// TIA Portal V20 export
DATA_BLOCK "DB_GestionSafetyGate"   // DB202
// stored: AutoNumber false, InstanceOfName FB_GestionSafetyGate, InstanceOfType FB
"FB_GestionSafetyGate"
   // VAR
   //    sExtGate { S7_SetPoint := 'True'} : "FB_CmdCylinder";
   //    sIntGate { S7_SetPoint := 'True'} : "FB_CmdCylinder";
   //    sExtGateCloseCmd : Bool;
   //    sExtGateOpenCmd : Bool;
   //    sIntGateCloseCmd : Bool;
   //    sIntGateOpenCmd : Bool;
   //    sJOG_Cmd : Bool;
   //    sRT_RefCmd : R_TRIG;
   //    sFT_RefCmd : F_TRIG;
   //    sExtGateOpenReq : Bool;
   //    sIntGateOpenReq : Bool;
   //    sExtGateOpened : Bool;
   //    sExtGateClosed : Bool;
   //    sIntGateOpened : Bool;
   //    sIntGateClosed : Bool;
   //    sWaitCloseShutterBeforeOpen : Bool;
   //    sWaitOpenShutterAfterClose : Bool;
   //    sTimeoutOpenCloseGateTimer : TON_TIME;
   //    sRT_IntGateOpenbyHMI { S7_SetPoint := 'True'} : R_TRIG;
   //    sFT_IntGateOpenbyHMI { S7_SetPoint := 'True'} : F_TRIG;
   //    sRT_ExtGateOpenbyHMI { S7_SetPoint := 'True'} : R_TRIG;
   //    sFT_ExtGateOpenbyHMI { S7_SetPoint := 'True'} : F_TRIG;
   //    sRT_ExtGateClose { S7_SetPoint := 'True'} : R_TRIG;
   //    sRT_ExtGateOpen { S7_SetPoint := 'True'} : R_TRIG;
   //    sRT_IntGateClose { S7_SetPoint := 'True'} : R_TRIG;
   //    sRT_IntGateOpen { S7_SetPoint := 'True'} : R_TRIG;
   //    sInterlockExtGateClose { S7_SetPoint := 'True'} : Bool;
   //    sInterlockExtGateOpen { S7_SetPoint := 'True'} : Bool;
   //    sInterlockIntGateClose : Bool;
   //    sInterlockIntGateOpen : Bool;
   // END_VAR
BEGIN
END_DATA_BLOCK
